{attribute addProperty BoxType "AMP8000-0030-0103-0103"}
{attribute addProperty Id "FSoE_Slave_Connection_1_Slave_MessageFSoE_Slave_Connection_1_Slave_Message_F5213E17567Standard_InputdataStandard_Inputdata_15EE41EA81FSLOGIC_InputsFSLOGIC_Inputs_0A35D0F1162FSoE_Slave_Connection_1_Master_MessageFSoE_Slave_Connection_1_Master_Message_79E02C6E567Standard_OutputdataStandard_Outputdata_3494233F81FSLOGIC_OutputsFSLOGIC_Outputs_49BC2EB9162"}
{attribute addProperty CRC "2943467165"}
{attribute addProperty SizeInBites "160"}
{attribute addProperty SizeInBytes "20"}
TYPE Device_Safety_AF71BE9D :
STRUCT
	{attribute addProperty Name "FSoE_Slave_Connection_1_Slave_Message"}
	FSoE_Slave_Connection_1_Slave_Message  : FSoE_Slave_Connection_1_Slave_Message_F5213E17;
	{attribute addProperty Name "Standard_Inputdata"}
	Standard_Inputdata  : Standard_Inputdata_15EE41EA;
	{attribute addProperty Name "FSLOGIC_Inputs"}
	FSLOGIC_Inputs  : FSLOGIC_Inputs_0A35D0F1;
	{attribute addProperty Name "FSoE_Slave_Connection_1_Master_Message"}
	FSoE_Slave_Connection_1_Master_Message  : FSoE_Slave_Connection_1_Master_Message_79E02C6E;
	{attribute addProperty Name "Standard_Outputdata"}
	Standard_Outputdata  : Standard_Outputdata_3494233F;
	{attribute addProperty Name "FSLOGIC_Outputs"}
	FSLOGIC_Outputs  : FSLOGIC_Outputs_49BC2EB9;
END_STRUCT
END_TYPE

(* stored: Version 1.2.0.0, ProductVersion 3.1.4024.9
   DUT Device_Safety_AF71BE9D: Id {8c9e7f95-0726-49a5-99d1-34fe2e8aac39} *)
